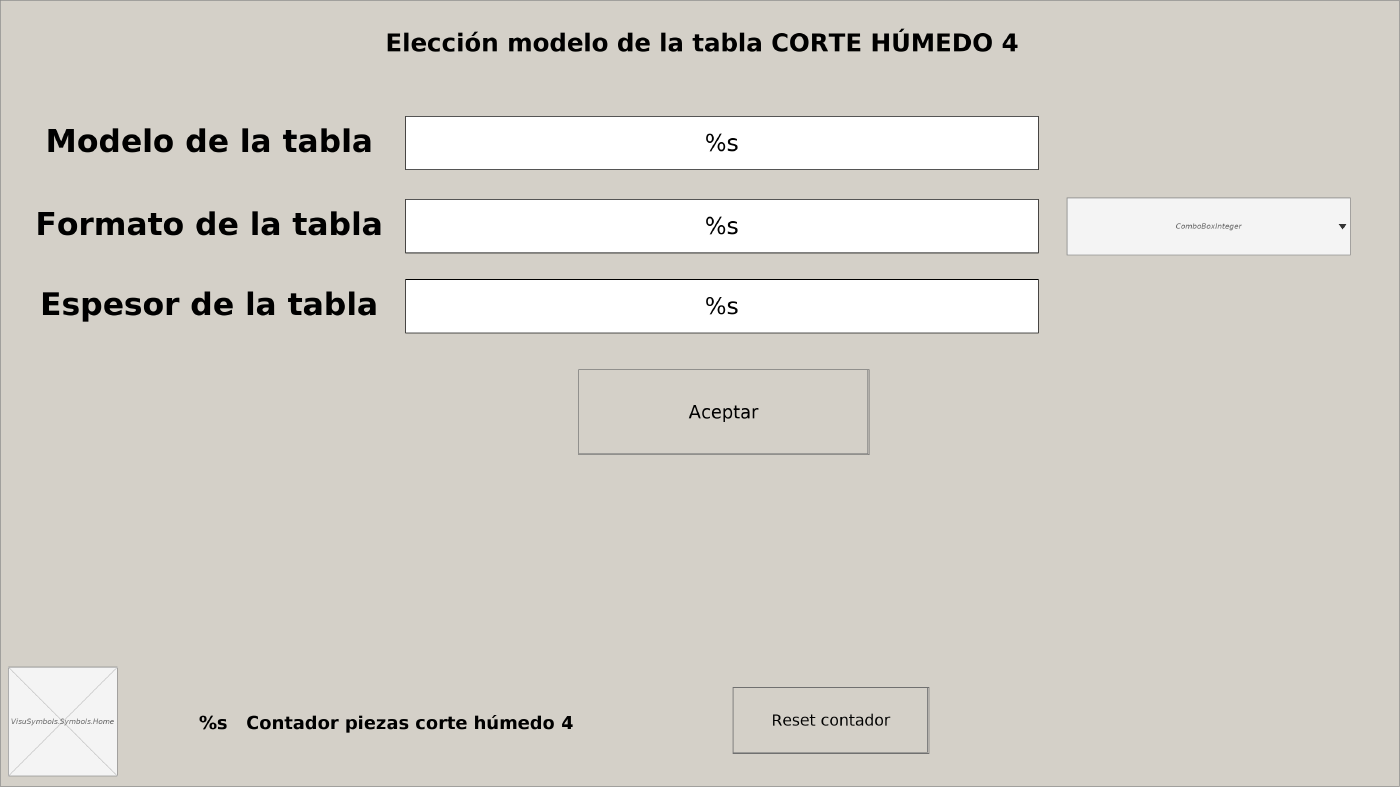
VISUALIZATION Modelo_Tabla_Ch4  // 1920x1080
    Label (36,136 517x115), "Modelo de la tabla"
    Rectangle (556,159 868x74), "%s", text variable: FuncParoNodoCorteH4Remote1.FunGeneCortHum4.s_ModeloEleccionTabla
        OnMouseDown: write the text variable via Edit
    Button (793,507 399x117), "Aceptar"
        tap FuncParoNodoCorteH4Remote1.FunGeneCortHum4.P_EscribirModelo
        OnMouseDown: change screen: Home_CortH4
    Label (439,29 1048x59), "Elección modelo de la tabla CORTE HÚMEDO 4"
    Rectangle (270,963 690x58), "%s Contador piezas corte húmedo 4", text variable: FuncParoNodoCorteH4Remote1.CortHum4StrFuncParoEnviar.Cont_Piezas
    Button (1005,943 269x91), "Reset contador"
        tap FuncParoNodoCorteH4Remote1.Funci_CortHum4.ResetContPiez
    Label (36,250 517x115), "Formato de la tabla"
    Rectangle (556,273 868x74), "%s", text variable: FuncParoNodoCorteH4Remote1.FunGeneCortHum4.s_FormatoEleccionTabla, input disabled if: FuncParoNodoCorteH4Remote1.FunGeneCortHum4.IndexListFormatoTabla<>6
        OnMouseUp: write the text variable via Edit
    Label (36,360 517x115), "Espesor de la tabla"
    Rectangle (556,383 868x74), "%s", text variable: FuncParoNodoCorteH4Remote1.FunGeneCortHum4.s_EspesorEleccionTabla
        OnMouseDown: write the text variable via Edit
    Image (11,915 150x150), image: VisuSymbols.Symbols.Home
        OnMouseClick: change screen: Home_CortH4
    ComboBoxInteger (1463,271 389x79), variable: FuncParoNodoCorteH4Remote1.FunGeneCortHum4.IndexListFormatoTabla, text list: 'FormatoTabla'
END_VISUALIZATION

(* stored: Version 1.1.0.1, ProductVersion 3.1.4024.12
   Visu Modelo_Tabla_Ch4: Id {80a4b618-84b7-4e17-b8f6-ff374c3b94b8} *)
